TYPE E_MFCS_Channel :
(
	BEGIN_CHANNEL,
	AM,
	SPOC,
	LOGGING,
	CM,
	CHANNEL_1,
	CHANNEL_2,
	CHANNEL_3,
	CHANNEL_4,
	CHANNEL_5,
	CHANNEL_6,
	CHANNEL_7,
	END_CHANNEL
);
END_TYPE

(* stored: Version 1.1.0.1, ProductVersion 3.1.4022.12
   DUT E_MFCS_Channel: Id {02762a82-a096-491e-8e93-cd36ce1faee7} *)
